PROGRAM MAIN_VISION
VAR
END_VAR


camera(dims := dimDist);

END_PROGRAM

(* stored: Version 1.1.0.1, ProductVersion 3.1.4024.6
   POU MAIN_VISION: Id {5ff15b36-f021-499b-8329-ff747c43ab93}, SpecialFunc None *)
